// TIA Portal V18 export
// export: Created 2025-12-01T17:53:03.178219Z, ExportSetting None, DisplayName Totally Integrated Automation Portal, DisplayVersion V18 Update 5, DisplayName TIA Portal Openness, DisplayVersion V18 Update 5, DisplayName TIA Portal Teamcenter Gateway, DisplayVersion V18, DisplayName TIA Portal Version Control Interface, DisplayVersion V18, DisplayName STEP 7 Professional, DisplayVersion V18 Update 5, DisplayName STEP 7 Safety, DisplayVersion V18, DisplayName WinCC Professional, DisplayVersion V18 Update 5
Screen "258 Scanner_807A1"  1280x800, Number=258, Template=02ManualUnit1
  ScreenLayer "Layer_0"
    FaceplateInstance "RCS_fpKeyenceSR1000_TP1200_1" at 10,129 size 1134x421  FaceplateTypeName=KeyenceSR1000@$@03_FacePlate@$@RCS_fpKeyenceSR1000_TP1200 V 0.0.6
      InterfacePropertyText "文本"  Text="807A1_Robot_3_Scan"
      Property := KeyenceSR1000Ctrl_807A1DB_sHMI
    Button "btnMenu8_7" at 1024,725 size 128x75  TextOff="F-读码器 807A1 / F-CodeReader 807A1 / Svetla", TextOn="F-读码器 807A1 / F-CodeReader 807A1"
      RangeAppearanceAnimation "RangeAppearanceAnimation"
        tag 
        0..0: back #636571, fore #000000
        1..1: back #0000ff, fore #000000
      on Click: ActivateScreen(Screen name := , Object number := 0)
    Button "按钮_9" at 128,725 size 128x75  PictureOff=向右箭头_0, TextOff="F-气缸1 / F-Cylinder 1", TextOn="F-气缸1 / F-Cylinder 1"
      on Click: ActivateScreen(Screen name := 250_Cylinder_F1, Object number := 0)
    Button "btnMenu4" at 384,725 size 128x75  TextOff="F-读码器 805A1 / F-CodeReader 805A1", TextOn="F-读码器 805A1 / F-CodeReader 805A1"
      on Click: ActivateScreen(Screen name := 252 Scanner_805A1, Object number := 0)
    Button "btnMenu5" at 512,725 size 128x75  TextOff="F-气缸2 / F-Cylinder 2", TextOn="F-气缸2 / F-Cylinder 2"
      on Click: ActivateScreen(Screen name := 253_Cylinder_F2, Object number := 0)
    Button "btnMenu6" at 640,725 size 128x75  TextOff="F-机器人2 / F-Robot2", TextOn="F-机器人2 / F-Robot2"
      on Click: ActivateScreen(Screen name := 254  Robot_2, Object number := 0)
    Button "按钮_1" at 896,725 size 128x75  TextOff="F-机器人3 / F-Robot3", TextOn="F-机器人3 / F-Robot3"
      on Click: ActivateScreen(Screen name := 257  Robot_3, Object number := 0)
    Button "btnMenu8_2" at 768,725 size 128x75  TextOff="F-气缸3 / F-Cylinder3", TextOn="F-气缸3 / F-Cylinder3"
      on Click: ActivateScreen(Screen name := 256_Cylinder_F3, Object number := 0)
    Button "btnMenu4_3" at 256,725 size 128x75  TextOff="F-机器人1 / F-Robot1", TextOn="F-机器人1 / F-Robot1"
      on Click: ActivateScreen(Screen name := 251  Robot_1, Object number := 0)
